KUKA KRL data list: Mill_FrameAut3.dat

&ACCESS RVP1
&REL 1
DEFDAT Mill_FrameAut3

   ;Amount of screw holes
   DECL CONST INT iScrewSize = 7

   ;Amount of pockets
   DECL CONST INT iPocketSize = 3

ENDDAT
